(* CODESYS project Codesys_Simulation.project

Project tree, tasks and I/O mapping:
  Device : CODESYS Control Win V3, 3S - Smart Software Solutions GmbH, order no. 305021, version 3.5.9.10
    application Application
      libraries: Standard, * (System)
      task MainTask (cyclic, interval t#20ms, priority 1) calls PLC_PRG
      program PLC_PRG [ST]
      Symbols
  libraries: VisuSymbols, 3.5.8.0 (System)
  visualisation Visualization
  text list GlobalTextList
  global variables GVL
*)

// GVL
VAR_GLOBAL

    (* ======================================== *)
    (* VARIABLES INDIVIDUALES — no borrar       *)
    (* ======================================== *)
    Q_VENTOSA_OMEGA  : BOOL;   (* Bit 0 → 1K1 *)
    Q_VENTOSA_PALET  : BOOL;   (* Bit 1 → 1K2 *)
    Q_LED_C1         : BOOL;   (* Bit 2 → 1K3 *)
    Q_LED_C2         : BOOL;   (* Bit 3 → 1K4 *)
    Q_LED_C3         : BOOL;   (* Bit 4 → 1K5 *)
    Q_LED_C4         : BOOL;   (* Bit 5 → 1K6 *)
    Q_LED_C5         : BOOL;   (* Bit 6 → 1K7 *)
    Q_LED_C6         : BOOL;   (* Bit 7 → 1K8 *)

    Q_START          : BOOL;   (* Bit 2 Puerto 2 *)
    Q_STOP           : BOOL;   (* Bit 3 Puerto 2 *)
    Q_EMERGENCIA     : BOOL;   (* Bit 4 Puerto 2 *)

    (* ======================================== *)
    (* BYTES DE SALIDA → FluidSIM              *)
    (* Construidos desde las variables arriba  *)
    (* ======================================== *)
    PUERTO_1         : BYTE;   (* → EasyPort1.InputPort1 *)
    PUERTO_2         : BYTE;   (* → EasyPort2.InputPort2 *)

    (* ======================================== *)
    (* CONTROL INTERNO                          *)
    (* ======================================== *)
    START            : BOOL;
    STOP             : BOOL;
    EMERGENCIA       : BOOL;
    SISTEMA_ACTIVO   : BOOL;

END_VAR

// Device/Application/PLC_PRG
PROGRAM PLC_PRG
VAR
    TEST_VENTOSA_OMEGA : BOOL;
    TEST_VENTOSA_PALET : BOOL;
    rStart             : R_TRIG;
    rStop              : R_TRIG;
END_VAR

rStart(CLK := GVL.START);
rStop(CLK  := GVL.STOP);

(* ======================================== *)
(* START / STOP / EMERGENCIA               *)
(* ======================================== *)

IF GVL.EMERGENCIA THEN
    GVL.SISTEMA_ACTIVO    := FALSE;
    TEST_VENTOSA_OMEGA    := FALSE;
    TEST_VENTOSA_PALET    := FALSE;
    GVL.Q_EMERGENCIA      := TRUE;
    GVL.Q_START           := FALSE;
    GVL.Q_STOP            := FALSE;

ELSIF rStop.Q THEN
    GVL.SISTEMA_ACTIVO    := FALSE;
    GVL.Q_START           := FALSE;
    GVL.Q_STOP            := TRUE;
    GVL.Q_EMERGENCIA      := FALSE;

ELSIF rStart.Q THEN
    GVL.SISTEMA_ACTIVO    := TRUE;
    GVL.Q_START           := TRUE;
    GVL.Q_STOP            := FALSE;
    GVL.Q_EMERGENCIA      := FALSE;
END_IF;

(* ======================================== *)
(* VENTOSAS — forzado manual de prueba     *)
(* ======================================== *)

IF GVL.SISTEMA_ACTIVO AND NOT GVL.EMERGENCIA THEN
    GVL.Q_VENTOSA_OMEGA := TEST_VENTOSA_OMEGA;
    GVL.Q_VENTOSA_PALET := TEST_VENTOSA_PALET;
ELSE
    GVL.Q_VENTOSA_OMEGA := FALSE;
    GVL.Q_VENTOSA_PALET := FALSE;
END_IF;

(* ======================================== *)
(* LEDs todos TRUE para prueba             *)
(* ======================================== *)

GVL.Q_LED_C1 := TRUE;
GVL.Q_LED_C2 := TRUE;
GVL.Q_LED_C3 := TRUE;
GVL.Q_LED_C4 := TRUE;
GVL.Q_LED_C5 := TRUE;
GVL.Q_LED_C6 := TRUE;

(* ======================================== *)
(* CONSTRUIR PUERTO_1 desde variables      *)
(* FluidSIM lee este BYTE completo         *)
(* ======================================== *)

GVL.PUERTO_1.0 := GVL.Q_VENTOSA_OMEGA;
GVL.PUERTO_1.1 := GVL.Q_VENTOSA_PALET;
GVL.PUERTO_1.2 := GVL.Q_LED_C1;
GVL.PUERTO_1.3 := GVL.Q_LED_C2;
GVL.PUERTO_1.4 := GVL.Q_LED_C3;
GVL.PUERTO_1.5 := GVL.Q_LED_C4;
GVL.PUERTO_1.6 := GVL.Q_LED_C5;
GVL.PUERTO_1.7 := GVL.Q_LED_C6;

(* ======================================== *)
(* CONSTRUIR PUERTO_2 desde variables      *)
(* ======================================== *)

GVL.PUERTO_2.2 := GVL.Q_START;
GVL.PUERTO_2.3 := GVL.Q_STOP;
GVL.PUERTO_2.4 := GVL.Q_EMERGENCIA;

END_PROGRAM

// /Visualization
VISUALIZATION Visualization  // 2x2
END_VISUALIZATION
